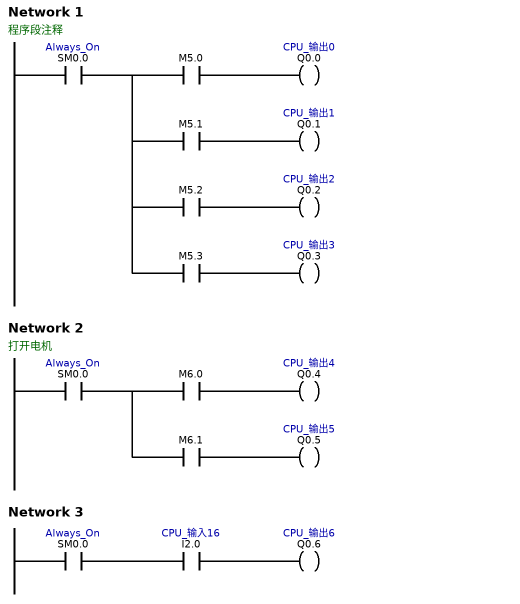
[picture p24: SBR12 networks 1-3]
Network 1
// 程序段注释
LD     Always_On:SM0.0
LPS
A      M5.0
=      CPU_输出0:Q0.0
LRD
A      M5.1
=      CPU_输出1:Q0.1
LRD
A      M5.2
=      CPU_输出2:Q0.2
LPP
A      M5.3
=      CPU_输出3:Q0.3
Network 2
// 打开电机
LD     Always_On:SM0.0
LPS
A      M6.0
=      CPU_输出4:Q0.4
LPP
A      M6.1
=      CPU_输出5:Q0.5
Network 3
LD     Always_On:SM0.0
A      CPU_输入16:I2.0
=      CPU_输出6:Q0.6
END_SUBROUTINE_BLOCK
